PROGRAM pConfig
VAR
	a: INT;
END_VAR

(*Configuracion Entradas y Salidas*)

_14_Config_Consum();
_00_Config_General();
_00_Config_PE();
_09_Config_CPump();
_05_Config_Drain();
_04_Config_Fill();
_06_Config_LEVEL();
_07_Config_Overflow();
_03_Config_PRESS();
_01_Config_SEG();
_02_Config_TEMP();
_10_Config_TK1();
_11_Config_TK2();
_15_Config_Winch();

pIO();

UPS();

END_PROGRAM

(* stored: Version 1.1.0.1, ProductVersion 3.1.4024.10
   POU pConfig: Id {2c3f7d8a-30b7-4862-a5f6-252ffa676804}, SpecialFunc None *)
